(* IEC 61131-3 sources: mocks/src/System/Timer, 11 files *)

(* ---- ConfigurableOffDelayMock.st ---- *)
NAMESPACE Simatic.Ax.Mocks
    /// Configurable Timer Mock for System.Timer.OffDelay - up to 4 timer instances
    /// Uses payload to configure individual timer states
    /// Timers are identified by call order (instance counter)
    FUNCTION_BLOCK ConfigurableOffDelayMock
        VAR_INPUT
            duration : LTIME;       // Preset duration
            signal : BOOL;          // Input signal
        END_VAR
        VAR_OUTPUT
            output : BOOL;          // Output
            elapsedTime : LTIME;    // Elapsed time
        END_VAR
        VAR_TEMP
            state : REF_TO ConfigurableOffDelayMockPayload;
        END_VAR

        // Get payload configuration
        state ?= AxUnit.Mocking.GetPayload();

        IF state = NULL THEN
            // Fallback if no payload is provided
            output := FALSE;
            elapsedTime := LTIME#0ms;
            RETURN;
        END_IF;

        // Increment call counter to identify timer instance
        state^.CallCounter := state^.CallCounter + 1;

        // Match timer by call order and apply configured state
        IF state^.CallCounter = 1 AND state^.T1_Enabled THEN
            output := state^.T1_Output;
            elapsedTime := state^.T1_ElapsedTime;
        ELSIF state^.CallCounter = 2 AND state^.T2_Enabled THEN
            output := state^.T2_Output;
            elapsedTime := state^.T2_ElapsedTime;
        ELSIF state^.CallCounter = 3 AND state^.T3_Enabled THEN
            output := state^.T3_Output;
            elapsedTime := state^.T3_ElapsedTime;
        ELSIF state^.CallCounter = 4 AND state^.T4_Enabled THEN
            output := state^.T4_Output;
            elapsedTime := state^.T4_ElapsedTime;
        ELSE
            // No matching timer configuration or counter overflow
            output := FALSE;
            elapsedTime := LTIME#0ms;
        END_IF;

    END_FUNCTION_BLOCK

    /// Payload configuration for ConfigurableOffDelayMock
    /// Allows configuration of up to 4 OffDelay timer instances
    /// Timers are identified by their call order (1st call = T1, 2nd call = T2, etc.)
    CLASS ConfigurableOffDelayMockPayload IMPLEMENTS AxUnit.Mocking.IPayload
        VAR PUBLIC
            // Internal call counter to track timer instances
            CallCounter : INT := 0;             // Tracks which timer instance is being called

            // Timer 1 configuration (1st timer call)
            T1_Enabled : BOOL := FALSE;         // Enable Timer 1
            T1_Output : BOOL := FALSE;          // Desired output for Timer 1
            T1_ElapsedTime : LTIME := LTIME#0ms; // Elapsed time for Timer 1

            // Timer 2 configuration (2nd timer call)
            T2_Enabled : BOOL := FALSE;         // Enable Timer 2
            T2_Output : BOOL := FALSE;          // Desired output for Timer 2
            T2_ElapsedTime : LTIME := LTIME#0ms; // Elapsed time for Timer 2

            // Timer 3 configuration (3rd timer call)
            T3_Enabled : BOOL := FALSE;         // Enable Timer 3
            T3_Output : BOOL := FALSE;          // Desired output for Timer 3
            T3_ElapsedTime : LTIME := LTIME#0ms; // Elapsed time for Timer 3

            // Timer 4 configuration (4th timer call)
            T4_Enabled : BOOL := FALSE;         // Enable Timer 4
            T4_Output : BOOL := FALSE;          // Desired output for Timer 4
            T4_ElapsedTime : LTIME := LTIME#0ms; // Elapsed time for Timer 4
        END_VAR

        /// Reset call counter - call this before each test cycle
        METHOD PUBLIC ResetCounter
            CallCounter := 0;
        END_METHOD
    END_CLASS
END_NAMESPACE

(* ---- ConfigurableOnDelayMock.st ---- *)
NAMESPACE Simatic.Ax.Mocks
    /// Configurable Timer Mock for System.Timer.OnDelay - up to 4 timer instances
    /// Uses payload to configure individual timer states
    /// Timers are identified by call order (instance counter)
    FUNCTION_BLOCK ConfigurableOnDelayMock
        VAR_INPUT
            duration : LTIME;       // Preset duration
            signal : BOOL;          // Input signal
        END_VAR
        VAR_OUTPUT
            output : BOOL;          // Output
            elapsedTime : LTIME;    // Elapsed time
        END_VAR
        VAR_TEMP
            state : REF_TO ConfigurableOnDelayMockPayload;
        END_VAR

        // Get payload configuration
        state ?= AxUnit.Mocking.GetPayload();

        IF state = NULL THEN
            // Fallback if no payload is provided
            output := FALSE;
            elapsedTime := LTIME#0ms;
            RETURN;
        END_IF;

        // Increment call counter to identify timer instance
        state^.CallCounter := state^.CallCounter + 1;

        // Match timer by call order and apply configured state
        IF state^.CallCounter = 1 AND state^.T1_Enabled THEN
            output := state^.T1_Output;
            elapsedTime := state^.T1_ElapsedTime;
        ELSIF state^.CallCounter = 2 AND state^.T2_Enabled THEN
            output := state^.T2_Output;
            elapsedTime := state^.T2_ElapsedTime;
        ELSIF state^.CallCounter = 3 AND state^.T3_Enabled THEN
            output := state^.T3_Output;
            elapsedTime := state^.T3_ElapsedTime;
        ELSIF state^.CallCounter = 4 AND state^.T4_Enabled THEN
            output := state^.T4_Output;
            elapsedTime := state^.T4_ElapsedTime;
        ELSE
            // No matching timer configuration or counter overflow
            output := FALSE;
            elapsedTime := LTIME#0ms;
        END_IF;

    END_FUNCTION_BLOCK

    /// Payload configuration for ConfigurableOnDelayMock
    /// Allows configuration of up to 4 OnDelay timer instances
    /// Timers are identified by their call order (1st call = T1, 2nd call = T2, etc.)
    CLASS ConfigurableOnDelayMockPayload IMPLEMENTS AxUnit.Mocking.IPayload
        VAR PUBLIC
            // Internal call counter to track timer instances
            CallCounter : INT := 0;             // Tracks which timer instance is being called

            // Timer 1 configuration (1st timer call)
            T1_Enabled : BOOL := FALSE;         // Enable Timer 1
            T1_Output : BOOL := FALSE;          // Desired output for Timer 1
            T1_ElapsedTime : LTIME := LTIME#0ms; // Elapsed time for Timer 1

            // Timer 2 configuration (2nd timer call)
            T2_Enabled : BOOL := FALSE;         // Enable Timer 2
            T2_Output : BOOL := FALSE;          // Desired output for Timer 2
            T2_ElapsedTime : LTIME := LTIME#0ms; // Elapsed time for Timer 2

            // Timer 3 configuration (3rd timer call)
            T3_Enabled : BOOL := FALSE;         // Enable Timer 3
            T3_Output : BOOL := FALSE;          // Desired output for Timer 3
            T3_ElapsedTime : LTIME := LTIME#0ms; // Elapsed time for Timer 3

            // Timer 4 configuration (4th timer call)
            T4_Enabled : BOOL := FALSE;         // Enable Timer 4
            T4_Output : BOOL := FALSE;          // Desired output for Timer 4
            T4_ElapsedTime : LTIME := LTIME#0ms; // Elapsed time for Timer 4
        END_VAR

        /// Reset call counter - call this before each test cycle
        METHOD PUBLIC ResetCounter
            CallCounter := 0;
        END_METHOD
    END_CLASS
END_NAMESPACE

(* ---- ConfigurableTimerMock.st ---- *)
NAMESPACE Simatic.Ax.Mocks
    /// Configurable Timer Mock for up to 4 timer instances
    /// Uses payload to configure individual timer states
    /// Can be used for both OnDelay and OffDelay timers
    /// Timers are identified by call order (instance counter)
    FUNCTION_BLOCK ConfigurableTimerMock
        VAR_INPUT
            duration : LTIME;       // Preset duration
            signal : BOOL;          // Input signal
        END_VAR
        VAR_OUTPUT
            output : BOOL;          // Output
            elapsedTime : LTIME;    // Elapsed time
        END_VAR
        VAR_TEMP
            state : REF_TO ConfigurableTimerMockPayload;
        END_VAR

        // Get payload configuration
        state ?= AxUnit.Mocking.GetPayload();

        IF state = NULL THEN
            // Fallback if no payload is provided
            output := FALSE;
            elapsedTime := LTIME#0ms;
            RETURN;
        END_IF;

        // Increment call counter to identify timer instance
        state^.CallCounter := state^.CallCounter + 1;

        // Match timer by call order and apply configured state
        IF state^.CallCounter = 1 AND state^.T1_Enabled THEN
            output := state^.T1_Output;
            elapsedTime := state^.T1_ElapsedTime;
        ELSIF state^.CallCounter = 2 AND state^.T2_Enabled THEN
            output := state^.T2_Output;
            elapsedTime := state^.T2_ElapsedTime;
        ELSIF state^.CallCounter = 3 AND state^.T3_Enabled THEN
            output := state^.T3_Output;
            elapsedTime := state^.T3_ElapsedTime;
        ELSIF state^.CallCounter = 4 AND state^.T4_Enabled THEN
            output := state^.T4_Output;
            elapsedTime := state^.T4_ElapsedTime;
        ELSE
            // No matching timer configuration or counter overflow
            output := FALSE;
            elapsedTime := LTIME#0ms;
        END_IF;

    END_FUNCTION_BLOCK

    /// Payload configuration for ConfigurableTimerMock
    /// Allows configuration of up to 4 timer instances
    /// Timers are identified by their call order (1st call = T1, 2nd call = T2, etc.)
    CLASS ConfigurableTimerMockPayload IMPLEMENTS AxUnit.Mocking.IPayload
        VAR PUBLIC
            // Internal call counter to track timer instances
            CallCounter : INT := 0;             // Tracks which timer instance is being called

            // Timer 1 configuration (1st timer call)
            T1_Enabled : BOOL := FALSE;         // Enable Timer 1
            T1_Output : BOOL := FALSE;          // Desired output for Timer 1
            T1_ElapsedTime : LTIME := LTIME#0ms; // Elapsed time for Timer 1

            // Timer 2 configuration (2nd timer call)
            T2_Enabled : BOOL := FALSE;         // Enable Timer 2
            T2_Output : BOOL := FALSE;          // Desired output for Timer 2
            T2_ElapsedTime : LTIME := LTIME#0ms; // Elapsed time for Timer 2

            // Timer 3 configuration (3rd timer call)
            T3_Enabled : BOOL := FALSE;         // Enable Timer 3
            T3_Output : BOOL := FALSE;          // Desired output for Timer 3
            T3_ElapsedTime : LTIME := LTIME#0ms; // Elapsed time for Timer 3

            // Timer 4 configuration (4th timer call)
            T4_Enabled : BOOL := FALSE;         // Enable Timer 4
            T4_Output : BOOL := FALSE;          // Desired output for Timer 4
            T4_ElapsedTime : LTIME := LTIME#0ms; // Elapsed time for Timer 4
        END_VAR

        /// Reset call counter - call this before each test cycle
        METHOD PUBLIC ResetCounter
            CallCounter := 0;
        END_METHOD
    END_CLASS
END_NAMESPACE

(* ---- IdentifierBasedOffDelayMock.st ---- *)
NAMESPACE Simatic.Ax.Mocks
    /// Identifier-based Timer Mock for System.Timer.OffDelay - up to 4 timer instances
    /// Timers are identified by their call position
    /// This allows testing conditional timer usage without duration dependency
    FUNCTION_BLOCK IdentifierBasedOffDelayMock
        VAR_INPUT
            duration : LTIME;       // Preset duration
            signal : BOOL;          // Input signal
        END_VAR
        VAR_OUTPUT
            output : BOOL;          // Output
            elapsedTime : LTIME;    // Elapsed time
        END_VAR
        VAR_TEMP
            state : REF_TO IdentifierBasedOffDelayMockPayload;
            matched : BOOL;
        END_VAR

        // Get payload configuration
        state ?= AxUnit.Mocking.GetPayload();

        IF state = NULL THEN
            // Fallback if no payload is provided
            output := FALSE;
            elapsedTime := LTIME#0ms;
            RETURN;
        END_IF;

        // Increment call counter
        state^.CallCounter := state^.CallCounter + 1;

        // Store current call information for debugging
        state^.LastCallDuration := duration;
        state^.LastCallSignal := signal;

        matched := FALSE;

        // Check each timer configuration
        // Timer is matched if enabled AND call counter matches the configured call position
        IF state^.T1_Enabled AND state^.CallCounter = state^.T1_CallPosition THEN
            output := state^.T1_Output;
            elapsedTime := state^.T1_ElapsedTime;
            matched := TRUE;
        ELSIF state^.T2_Enabled AND state^.CallCounter = state^.T2_CallPosition THEN
            output := state^.T2_Output;
            elapsedTime := state^.T2_ElapsedTime;
            matched := TRUE;
        ELSIF state^.T3_Enabled AND state^.CallCounter = state^.T3_CallPosition THEN
            output := state^.T3_Output;
            elapsedTime := state^.T3_ElapsedTime;
            matched := TRUE;
        ELSIF state^.T4_Enabled AND state^.CallCounter = state^.T4_CallPosition THEN
            output := state^.T4_Output;
            elapsedTime := state^.T4_ElapsedTime;
            matched := TRUE;
        END_IF;

        // Default if no match found
        IF NOT matched THEN
            output := FALSE;
            elapsedTime := LTIME#0ms;
        END_IF;

    END_FUNCTION_BLOCK

    /// Payload configuration for IdentifierBasedOffDelayMock
    /// Each timer is configured with its expected call position
    /// This allows flexible testing of conditional timer logic
    CLASS IdentifierBasedOffDelayMockPayload IMPLEMENTS AxUnit.Mocking.IPayload
        VAR PUBLIC
            // Internal call counter
            CallCounter : INT := 0;               // Tracks current call number

            // Debug information
            LastCallDuration : LTIME := LTIME#0ms;  // Last called duration
            LastCallSignal : BOOL := FALSE;         // Last called signal

            // Timer 1 configuration
            T1_Enabled : BOOL := FALSE;           // Enable Timer 1
            T1_CallPosition : INT := 1;           // Expected call position (1st, 2nd, 3rd, etc.)
            T1_Output : BOOL := FALSE;            // Desired output for Timer 1
            T1_ElapsedTime : LTIME := LTIME#0ms;  // Elapsed time for Timer 1

            // Timer 2 configuration
            T2_Enabled : BOOL := FALSE;           // Enable Timer 2
            T2_CallPosition : INT := 2;           // Expected call position
            T2_Output : BOOL := FALSE;            // Desired output for Timer 2
            T2_ElapsedTime : LTIME := LTIME#0ms;  // Elapsed time for Timer 2

            // Timer 3 configuration
            T3_Enabled : BOOL := FALSE;           // Enable Timer 3
            T3_CallPosition : INT := 3;           // Expected call position
            T3_Output : BOOL := FALSE;            // Desired output for Timer 3
            T3_ElapsedTime : LTIME := LTIME#0ms;  // Elapsed time for Timer 3

            // Timer 4 configuration
            T4_Enabled : BOOL := FALSE;           // Enable Timer 4
            T4_CallPosition : INT := 4;           // Expected call position
            T4_Output : BOOL := FALSE;            // Desired output for Timer 4
            T4_ElapsedTime : LTIME := LTIME#0ms;  // Elapsed time for Timer 4
        END_VAR

        /// Reset call counter - call this before each test cycle
        METHOD PUBLIC ResetCounter
            CallCounter := 0;
        END_METHOD
    END_CLASS
END_NAMESPACE

(* ---- IdentifierBasedOnDelayMock.st ---- *)
NAMESPACE Simatic.Ax.Mocks
    /// Identifier-based Timer Mock for System.Timer.OnDelay - up to 4 timer instances
    /// Timers are identified by their call position
    /// This allows testing conditional timer usage without duration dependency
    FUNCTION_BLOCK IdentifierBasedOnDelayMock
        VAR_INPUT
            duration : LTIME;       // Preset duration
            signal : BOOL;          // Input signal
        END_VAR
        VAR_OUTPUT
            output : BOOL;          // Output
            elapsedTime : LTIME;    // Elapsed time
        END_VAR
        VAR_TEMP
            state : REF_TO IdentifierBasedOnDelayMockPayload;
            matched : BOOL;
        END_VAR

        // Get payload configuration
        state ?= AxUnit.Mocking.GetPayload();

        IF state = NULL THEN
            // Fallback if no payload is provided
            output := FALSE;
            elapsedTime := LTIME#0ms;
            RETURN;
        END_IF;

        // Increment call counter
        state^.CallCounter := state^.CallCounter + 1;

        // Store current call information for debugging
        state^.LastCallDuration := duration;
        state^.LastCallSignal := signal;

        matched := FALSE;

        // Check each timer configuration
        // Timer is matched if enabled AND call counter matches the configured call position
        IF state^.T1_Enabled AND state^.CallCounter = state^.T1_CallPosition THEN
            output := state^.T1_Output;
            elapsedTime := state^.T1_ElapsedTime;
            matched := TRUE;
        ELSIF state^.T2_Enabled AND state^.CallCounter = state^.T2_CallPosition THEN
            output := state^.T2_Output;
            elapsedTime := state^.T2_ElapsedTime;
            matched := TRUE;
        ELSIF state^.T3_Enabled AND state^.CallCounter = state^.T3_CallPosition THEN
            output := state^.T3_Output;
            elapsedTime := state^.T3_ElapsedTime;
            matched := TRUE;
        ELSIF state^.T4_Enabled AND state^.CallCounter = state^.T4_CallPosition THEN
            output := state^.T4_Output;
            elapsedTime := state^.T4_ElapsedTime;
            matched := TRUE;
        END_IF;

        // Default if no match found
        IF NOT matched THEN
            output := FALSE;
            elapsedTime := LTIME#0ms;
        END_IF;

    END_FUNCTION_BLOCK

    /// Payload configuration for IdentifierBasedOnDelayMock
    /// Each timer is configured with its expected call position
    /// This allows flexible testing of conditional timer logic
    CLASS IdentifierBasedOnDelayMockPayload IMPLEMENTS AxUnit.Mocking.IPayload
        VAR PUBLIC
            // Internal call counter
            CallCounter : INT := 0;               // Tracks current call number

            // Debug information
            LastCallDuration : LTIME := LTIME#0ms;  // Last called duration
            LastCallSignal : BOOL := FALSE;         // Last called signal

            // Timer 1 configuration
            T1_Enabled : BOOL := FALSE;           // Enable Timer 1
            T1_CallPosition : INT := 1;           // Expected call position (1st, 2nd, 3rd, etc.)
            T1_Output : BOOL := FALSE;            // Desired output for Timer 1
            T1_ElapsedTime : LTIME := LTIME#0ms;  // Elapsed time for Timer 1

            // Timer 2 configuration
            T2_Enabled : BOOL := FALSE;           // Enable Timer 2
            T2_CallPosition : INT := 2;           // Expected call position
            T2_Output : BOOL := FALSE;            // Desired output for Timer 2
            T2_ElapsedTime : LTIME := LTIME#0ms;  // Elapsed time for Timer 2

            // Timer 3 configuration
            T3_Enabled : BOOL := FALSE;           // Enable Timer 3
            T3_CallPosition : INT := 3;           // Expected call position
            T3_Output : BOOL := FALSE;            // Desired output for Timer 3
            T3_ElapsedTime : LTIME := LTIME#0ms;  // Elapsed time for Timer 3

            // Timer 4 configuration
            T4_Enabled : BOOL := FALSE;           // Enable Timer 4
            T4_CallPosition : INT := 4;           // Expected call position
            T4_Output : BOOL := FALSE;            // Desired output for Timer 4
            T4_ElapsedTime : LTIME := LTIME#0ms;  // Elapsed time for Timer 4
        END_VAR

        /// Reset call counter - call this before each test cycle
        METHOD PUBLIC ResetCounter
            CallCounter := 0;
        END_METHOD
    END_CLASS
END_NAMESPACE

(* ---- IdentifierBasedTimerMock.st ---- *)
NAMESPACE Simatic.Ax.Mocks
    /// Identifier-based Timer Mock for up to 4 timer instances
    /// Timers are identified by a unique ID passed via a special mechanism
    /// This allows testing conditional timer usage without duration dependency
    FUNCTION_BLOCK IdentifierBasedTimerMock
        VAR_INPUT
            duration : LTIME;       // Preset duration
            signal : BOOL;          // Input signal
        END_VAR
        VAR_OUTPUT
            output : BOOL;          // Output
            elapsedTime : LTIME;    // Elapsed time
        END_VAR
        VAR_TEMP
            state : REF_TO IdentifierBasedTimerMockPayload;
            matched : BOOL;
        END_VAR

        // Get payload configuration
        state ?= AxUnit.Mocking.GetPayload();

        IF state = NULL THEN
            // Fallback if no payload is provided
            output := FALSE;
            elapsedTime := LTIME#0ms;
            RETURN;
        END_IF;

        // Increment call counter
        state^.CallCounter := state^.CallCounter + 1;

        // Store current call information for debugging
        state^.LastCallDuration := duration;
        state^.LastCallSignal := signal;

        matched := FALSE;

        // Check each timer configuration
        // Timer is matched if enabled AND call counter matches the configured call position
        IF state^.T1_Enabled AND state^.CallCounter = state^.T1_CallPosition THEN
            output := state^.T1_Output;
            elapsedTime := state^.T1_ElapsedTime;
            matched := TRUE;
        ELSIF state^.T2_Enabled AND state^.CallCounter = state^.T2_CallPosition THEN
            output := state^.T2_Output;
            elapsedTime := state^.T2_ElapsedTime;
            matched := TRUE;
        ELSIF state^.T3_Enabled AND state^.CallCounter = state^.T3_CallPosition THEN
            output := state^.T3_Output;
            elapsedTime := state^.T3_ElapsedTime;
            matched := TRUE;
        ELSIF state^.T4_Enabled AND state^.CallCounter = state^.T4_CallPosition THEN
            output := state^.T4_Output;
            elapsedTime := state^.T4_ElapsedTime;
            matched := TRUE;
        END_IF;

        // Default if no match found
        IF NOT matched THEN
            output := FALSE;
            elapsedTime := LTIME#0ms;
        END_IF;

    END_FUNCTION_BLOCK

    /// Payload configuration for IdentifierBasedTimerMock
    /// Each timer is configured with its expected call position
    /// This allows flexible testing of conditional timer logic
    CLASS IdentifierBasedTimerMockPayload IMPLEMENTS AxUnit.Mocking.IPayload
        VAR PUBLIC
            // Internal call counter
            CallCounter : INT := 0;               // Tracks current call number

            // Debug information
            LastCallDuration : LTIME := LTIME#0ms;  // Last called duration
            LastCallSignal : BOOL := FALSE;         // Last called signal

            // Timer 1 configuration
            T1_Enabled : BOOL := FALSE;           // Enable Timer 1
            T1_CallPosition : INT := 1;           // Expected call position (1st, 2nd, 3rd, etc.)
            T1_Output : BOOL := FALSE;            // Desired output for Timer 1
            T1_ElapsedTime : LTIME := LTIME#0ms;  // Elapsed time for Timer 1

            // Timer 2 configuration
            T2_Enabled : BOOL := FALSE;           // Enable Timer 2
            T2_CallPosition : INT := 2;           // Expected call position
            T2_Output : BOOL := FALSE;            // Desired output for Timer 2
            T2_ElapsedTime : LTIME := LTIME#0ms;  // Elapsed time for Timer 2

            // Timer 3 configuration
            T3_Enabled : BOOL := FALSE;           // Enable Timer 3
            T3_CallPosition : INT := 3;           // Expected call position
            T3_Output : BOOL := FALSE;            // Desired output for Timer 3
            T3_ElapsedTime : LTIME := LTIME#0ms;  // Elapsed time for Timer 3

            // Timer 4 configuration
            T4_Enabled : BOOL := FALSE;           // Enable Timer 4
            T4_CallPosition : INT := 4;           // Expected call position
            T4_Output : BOOL := FALSE;            // Desired output for Timer 4
            T4_ElapsedTime : LTIME := LTIME#0ms;  // Elapsed time for Timer 4
        END_VAR

        /// Reset call counter - call this before each test cycle
        METHOD PUBLIC ResetCounter
            CallCounter := 0;
        END_METHOD
    END_CLASS
END_NAMESPACE

(* ---- OffDelayMock_false.st ---- *)
NAMESPACE Simatic.Ax.Mocks
    /// Off-Delay Timer Mock - Always returns FALSE
    /// System.Timer interface (signal/duration)
    FUNCTION_BLOCK OffDelayMock_false
        VAR_INPUT
            duration : LTIME;       // Preset duration
            signal : BOOL;          // Input signal
        END_VAR
        VAR_OUTPUT
            output : BOOL;          // Output
            elapsedTime : LTIME;    // Elapsed time
        END_VAR
        output := FALSE;
        elapsedTime := LTIME#0ms;
    END_FUNCTION_BLOCK
END_NAMESPACE

(* ---- OffDelayMock_true.st ---- *)
NAMESPACE Simatic.Ax.Mocks
    /// Off-Delay Timer Mock - Always returns TRUE
    /// System.Timer interface (signal/duration)
    FUNCTION_BLOCK OffDelayMock_true
        VAR_INPUT
            duration : LTIME;       // Preset duration
            signal : BOOL;          // Input signal
        END_VAR
        VAR_OUTPUT
            output : BOOL;          // Output
            elapsedTime : LTIME;    // Elapsed time
        END_VAR
        output := TRUE;
        elapsedTime := duration;
    END_FUNCTION_BLOCK
END_NAMESPACE

(* ---- OnDelayMock_false.st ---- *)
NAMESPACE Simatic.Ax.Mocks
    /// On-Delay Timer Mock - Always returns FALSE
    /// System.Timer interface (signal/duration)
    FUNCTION_BLOCK OnDelayMock_false
        VAR_INPUT
            duration : LTIME;       // Preset duration
            signal : BOOL;          // Input signal
        END_VAR
        VAR_OUTPUT
            output : BOOL;          // Output
            elapsedTime : LTIME;    // Elapsed time
        END_VAR
        output := FALSE;
        elapsedTime := LTIME#0ms;
    END_FUNCTION_BLOCK
END_NAMESPACE

(* ---- OnDelayMock_true.st ---- *)
NAMESPACE Simatic.Ax.Mocks
    /// On-Delay Timer Mock - Always returns TRUE
    /// System.Timer interface (signal/duration)
    FUNCTION_BLOCK OnDelayMock_true
        VAR_INPUT
            duration : LTIME;       // Preset duration
            signal : BOOL;          // Input signal
        END_VAR
        VAR_OUTPUT
            output : BOOL;          // Output
            elapsedTime : LTIME;    // Elapsed time
        END_VAR
        output := TRUE;
        elapsedTime := duration;
    END_FUNCTION_BLOCK
END_NAMESPACE

(* ---- OnDelayMockWithTwoTimers.st ---- *)
NAMESPACE Simatic.Ax.Mocks
    /// This Mock can be used in Classes/FunctionBlocks where are two OnDelay instances are used
    {axcode:docs-v0:@simatic-ax/generators:OnDelayMockWithTwoTimers.md}
    FUNCTION_BLOCK OnDelayMock2Timer
        VAR_INPUT
            duration : LTIME;
            signal : BOOL;
        END_VAR
        VAR_OUTPUT
            output : BOOL;
            elapsedTime : LTIME;
        END_VAR
        VAR_TEMP
            state : REF_TO OnDelayMockState;
        END_VAR

        state ?= AxUnit.Mocking.GetPayload();
        output := TRUE;
        return;
        IF (signal = FALSE) THEN
            output := FALSE;
        ELSE
            IF duration = T#1s THEN
                output := state^.StatusTimer1;
            END_IF;
            IF duration = T#2s THEN
                output := state^.StatusTimer2 ;
            END_IF;
        END_IF;

    END_FUNCTION_BLOCK

    /// The returned states for the Timer1 and Timer2
    {axcode:docs-v0:@simatic-ax/generators:OnDelayMockWithTwoTimers.md}
    CLASS OnDelayMockState IMPLEMENTS AxUnit.Mocking.IPayload
        VAR PUBLIC
            StatusTimer1 : BOOL;
            StatusTimer2 : BOOL;
        END_VAR
    END_CLASS
END_NAMESPACE
